// TIA Portal V16 export
// export: Created 2022-11-17T15:49:39.2822426Z, ExportSetting WithDefaults, DisplayName Totally Integrated Automation Portal, DisplayVersion V16 Update 6, DisplayName TIA Portal Version Control Interface, DisplayVersion V16 Update 2, DisplayName TIA Portal Openness, DisplayVersion V16 Update 6, DisplayName SINAMICS Startdrive Advanced, DisplayVersion V16 Update 5, DisplayName SINAMICS Startdrive G130, G150, S120, S150, SINAMICS MV, S210, DisplayVersion V16 Update 5, DisplayName SINAMICS Startdrive G110M, G120, G120C, G120D, G120P, G115D, DisplayVersion V16 Update 5, DisplayName STEP 7 Professional, DisplayVersion V16 Update 6, DisplayName STEP 7 Safety, DisplayVersion V16, DisplayName WinCC Advanced, DisplayVersion V16 Update 6
DATA_BLOCK "DB21_DisplayGeneralData"   // DB21
{ S7_Optimized_Access := 'FALSE' }
AUTHOR : Robopac
VERSION : 0.0
// stored: AutoNumber false, IsOnlyStoredInLoadMemory false, IsWriteProtectedInAS false
   VAR RETAIN
      dbx0_0 : Bool := TRUE;   // Welder unit included(1)/excluded (Display-General Data)
      dbx0_1 : Bool := FALSE;   // Machine included(1)/excluded (Display-General Data)
      dbx0_2 : Bool := TRUE;   // Pallet load/unload included(1)/excluded (Display-Sysdata)
      dbx0_3 : Bool := TRUE;   // Load pallet with forklift selection by display (Display-Sysdata)
      dbx0_4 : Bool := TRUE;   // Unload pallet with forklift selection by display (Display-Sysdata)
      dbx0_5 : Bool := FALSE;
      dbx0_6 : Bool := TRUE;
      dbx0_7 : Bool := FALSE;
      dbb1 : Byte := 16#00;
      dbw2 : Int := 3;   // PLC SW major release
      dbw4 : Int := 0;   // PLC SW minor release
      dbw6 : Int := 90;   // Spool carriage upward for spring clamp at begin cycle (Display-General Data)
      dbw8 : Int := 0;   // Spool carriage downward for film tail at the cycle begin (Display-General Data)
      dbw10 : Int := 2;   // Film thickness (Display-General Data)
      dbw12 : Int := 700;   // Welding time (Display-General Data)
      dbw14 : Int := 0;   // Low speed for Helix conveyor movement (%) (Display-Sysdata)
      dbw16 : Int := 0;   // High speed for Helix conveyor movement (%) (Display-Sysdata)
      dbw18 : Int := 500;   // Delay on pallet positioning (Display-General Data)
      dbw20 : Int := 10000;   // Delay for load/unload pallet simultaneously (Display-General Data)
      dbw22 : Int := 100;   // Deceleration for pallet positioning (Display-General Data)
      dbw24 : Int := 1;   // Time for pallet load with forklift
      dbw26 : Int := 0;   // Override for ring movement in manul mode (Display-General Data)
      dbw28 : Int := 100;   // TIMER CICLO FIERA (attesa tra cicli successivi)
      dbw30 : Int := 0;   // Film prestretch for film prestretch test cycle (Display-General Data)
      dbw32 : Int := 0;   // Film prestretch increase for film prestretch test (Display-General Data)
      dbw34 : Int := 0;   // Film supplied every revolution for film prestretch test (Display-General Data)
      dbw36 : Int := 0;   // Time for spool carriage upward for table cycle (Display-Sysdata)
      dbw38 : Int := 2000;   // Time for spool carriage upward for table cycle (Display-Sysdata)
      dbw40 : Int := 15000;   // Time load with forklift
      dbw42 : Int := 10000;   // Time unload with forklift
   END_VAR
BEGIN
END_DATA_BLOCK
